FUNCTION_BLOCK FB_LensSetMock EXTENDS FB_FalliblePublicMock IMPLEMENTS I_LensSet
VAR
    afFocalLength : ARRAY [1..GVL_Physics.nMaxNumLensesInSet] OF LREAL;
    afbLensMock : ARRAY [1..GVL_Physics.nMaxNumLensesInSet] OF FB_LensMock;
    nNumLenses : INT;
END_VAR

METHOD GetLens
VAR_INPUT
    LensNum	: INT;
END_VAR
VAR_IN_OUT
    Lens	: FB_Lens;
END_VAR

Lens.Copy(afbLensMock[LensNum]);
END_METHOD


PROPERTY NumLenses : INT
GET

NumLenses := nNumLenses;
END_GET
SET

nNumLenses := NumLenses;
END_SET
END_PROPERTY


METHOD SetMaterialNameOf
VAR_INPUT
    LensNum	: INT;
    MaterialFormula : T_MaxString;
END_VAR

afbLensMock[LensNum].MaterialFormula := MaterialFormula;
END_METHOD


METHOD SetMultiplierOf
VAR_INPUT
    LensNum	: INT;
    Multiplier : INT;
END_VAR

afbLensMock[LensNum].Multiplier := Multiplier;
END_METHOD


METHOD SetRadiusOf
VAR_INPUT
    LensNum : INT;
    Radius : I_QuantityLREAL;
END_VAR

afbLensMock[LensNum].SetRadius(Radius);
END_METHOD


METHOD SetValid
VAR
    nIndex : INT;
END_VAR
VAR
    fbRadius : FB_QuantityLREALPublicMock;
END_VAR

ClearError();

fbRadius.Val := 1.0;
fbRadius.Units := 'm';

FOR nIndex := 1 TO GVL_Physics.nMaxNumLensesInSet BY 1 DO
    afbLensMock[nIndex].Multiplier := 1;
    afbLensMock[nIndex].SetRadius(fbRadius);
    afbLensMock[nIndex].MaterialFormula := 'Be';
END_FOR
END_METHOD

END_FUNCTION_BLOCK

(* stored: Version 1.1.0.1
   POU FB_LensSetMock: Id {81efb5ab-6e66-4093-a776-0c018358a642}, SpecialFunc None
   Method GetLens: Id {14bb5de5-7cf5-45f2-8b3c-d5e0518be57c}
   Property NumLenses: Id {0de8fc65-e8dc-4248-ab31-049f75250b77}
   Get Get: Id {9bca06c1-467c-4734-8686-595d1621e3e3}
   Set Set: Id {049e4945-30a7-44eb-aa9f-e85882a20364}
   Method SetMaterialNameOf: Id {37855da5-e9a8-4247-be85-98c220363308}
   Method SetMultiplierOf: Id {a2d3085f-8a83-4983-8c40-581e8915de41}
   Method SetRadiusOf: Id {ae316088-ffb3-4f48-8984-1fe3e09c2632}
   Method SetValid: Id {8028786d-6bf1-49c2-919b-77cc8caff0f8} *)
